{attribute 'qualified_only'}
{attribute 'strict'}
TYPE eBroach :
(
	Master	:= 0,
	V1		:= 2,
	V2		:= 3,
	V3		:= 4,
	V4		:= 5,
	V5		:= 6,
	V6		:= 7
);
END_TYPE

(* stored: Version 1.1.0.1, ProductVersion 3.1.4024.13
   DUT eBroach: Id {be260c27-60b9-4103-a70e-857e0ce3d49e} *)
